FUNCTION TryConvert_SINT_TO_REAL : BOOL
VAR_INPUT
	in : SINT;
	out : REFERENCE TO REAL;
END_VAR

out := SINT_TO_REAL(in);
TryConvert_SINT_TO_REAL := TRUE;

END_FUNCTION

(* stored: Version 1.1.0.1, ProductVersion 3.1.4024.12
   POU TryConvert_SINT_TO_REAL: Id {14542013-39ba-4c6d-9fdc-0a748b9f786d}, SpecialFunc None *)
